FUNCTION_BLOCK GroupStatus
VAR_INPUT
END_VAR
VAR_OUTPUT
END_VAR
VAR
    _Busy : BOOL;
    _Error : BOOL;
END_VAR

// Copyright (c) 2024 Loupe (https://loupe.team), provided under the MIT License.

METHOD Busy
VAR_INPUT
    Message : STRING[80];
END_VAR
// Copyright (c) 2024 Loupe (https://loupe.team), provided under the MIT License.

_Busy := TRUE;
END_METHOD

METHOD Error
VAR_INPUT
    Message : STRING[80];
END_VAR
// Copyright (c) 2024 Loupe (https://loupe.team), provided under the MIT License.

_Error := TRUE;
END_METHOD

PROPERTY IsBusy : BOOL
GET
// Copyright (c) 2024 Loupe (https://loupe.team), provided under the MIT License.

IsBusy := NOT _Error AND _Busy;
END_GET
END_PROPERTY

PROPERTY IsDone : BOOL
GET
// Copyright (c) 2024 Loupe (https://loupe.team), provided under the MIT License.

IsDone := NOT _Error AND NOT _Busy;
END_GET
END_PROPERTY

PROPERTY IsError : BOOL
GET
// Copyright (c) 2024 Loupe (https://loupe.team), provided under the MIT License.

IsError := _Error;
END_GET
END_PROPERTY

METHOD Ok : BOOL
VAR_INPUT
END_VAR
// Copyright (c) 2024 Loupe (https://loupe.team), provided under the MIT License.
END_METHOD

METHOD Reset
VAR_INPUT
END_VAR
// Copyright (c) 2024 Loupe (https://loupe.team), provided under the MIT License.

_Busy := FALSE;
_Error := FALSE;
END_METHOD

PROPERTY Status : PLCopenStatusBase
GET
// Copyright (c) 2024 Loupe (https://loupe.team), provided under the MIT License.

IF _Error THEN

    Status := PLCopenStatusBase.ERROR;

ELSIF _Busy THEN

    Status := PLCopenStatusBase.BUSY;

ELSE

    Status := PLCopenStatusBase.ERR_OK;

END_IF
END_GET
END_PROPERTY

END_FUNCTION_BLOCK

(* stored: Version 1.1.0.1
   POU GroupStatus: Id {64a0f666-997c-47bb-a11d-deccd3a678a8}, SpecialFunc None
   Method Busy: Id {fe61334e-f225-49f0-8a17-ff1b39f4d264}
   Method Error: Id {a774ec91-6e7f-4e7e-9619-0d714616bbff}
   Property IsBusy: Id {8b172ddf-04e9-4236-806d-134b8ae3c542}
   Get Get: Id {55a7db60-84c5-4687-ab04-0cf56c15f341}
   Property IsDone: Id {c0071902-5599-4ac5-a0b2-7e49d560bd64}
   Get Get: Id {dcf7e083-dee0-44d7-b7f1-f038315678db}
   Property IsError: Id {e4413f7f-b554-4b5c-8287-095be611bfa9}
   Get Get: Id {0593bd48-e708-4565-9399-9aa14aee0b35}
   Method Ok: Id {1be299bc-a77b-4303-b016-e012e735be40}
   Method Reset: Id {77e19edc-3ebc-48b1-879e-51ee30f840ea}
   Property Status: Id {34f306bb-0f78-474b-ae87-31c2cd249735}
   Get Get: Id {1ccbce53-2a69-4d36-bbbc-ebe695682689} *)
